(* CODESYS project IA_Lab-7.2.project

Project tree, tasks and I/O mapping:
  CAM tables/
  CNC programs/
  Data types/
  Global Variables/
    global variables Global_Variables
    global variables Variable_Configuration
  POUs/
    program PLC_PRG [LD]
  Visualizations/
  GlobalImagePool
*)

// Global Variables/Global_Variables
VAR_GLOBAL
END_VAR

// Global Variables/Variable_Configuration
VAR_CONFIG
END_VAR

// POUs/PLC_PRG
PROGRAM PLC_PRG
VAR
	A: BOOL;
	y: BOOL;
	C: CTU;
	ghhj: INT;
	Temp: BOOL;
	Reset: BOOL;
END_VAR

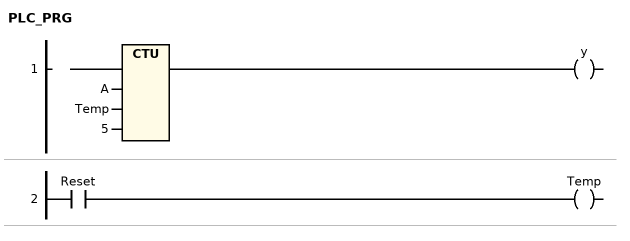
// NETWORK 1
y := CTU(A, Temp, 5);

// NETWORK 2
Temp := Reset;

END_PROGRAM
